FUNCTION_BLOCK Esp32EthernetKitIO (* Template for Modular IO with Esp32EthernetKit board *)
  (* Standard: 61499-2; Description: Copyright (c) 2024 Dirk O. Kaar This program and the accompanying materials are made available under the terms of the Eclipse Public License 2.0 which is available at https://www.eclipse.org/legal/epl-2.0/ SPDX-License-Identifier: EPL-2.0 *)
  (* Version 1.0, 2024-01-13, Dirk O. Kaar *)
  (* Version 3.0, 2025-04-14, Patrick Aigner, changed package *)
  PACKAGE eclipse4diac::io::zephyr;
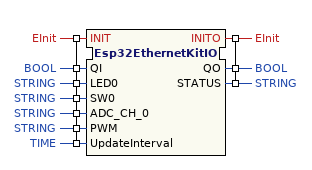
  EVENT_INPUT
    INIT : EInit WITH QI, UpdateInterval, LED0, SW0, ADC_CH_0, PWM; (* Service Initialization *)
  END_EVENT
  EVENT_OUTPUT
    INITO : EInit WITH QO, STATUS; (* Initialization Confirm *)
  END_EVENT
  VAR_INPUT
    QI : BOOL; (* Event Input Qualifier *)
    LED0 : STRING;
    SW0 : STRING;
    ADC_CH_0 : STRING;
    PWM : STRING;
    UpdateInterval : TIME := T#40ms; (* Update interval *)
  END_VAR
  VAR_OUTPUT
    QO : BOOL; (* Event Output Qualifier *)
    STATUS : STRING; (* Service Status *)
  END_VAR
  (* Service APPLICATION/RESOURCE: Template for Modular IO with Esp32EthernetKit board *)
END_FUNCTION_BLOCK
